INTERFACE I_Observable EXTENDS __SYSTEM.IQueryInterface

METHOD Attach : BOOL
VAR_INPUT
    ipObserver:         I_Observer;
END_VAR
END_METHOD

METHOD Detach : BOOL
VAR_INPUT
    ipObserver:         I_Observer;
END_VAR
END_METHOD

PROPERTY nObserverCount : UDINT
GET
END_GET
END_PROPERTY

METHOD Notify : I_Observable
VAR_INPUT
END_VAR
END_METHOD

METHOD NotifyLast : I_Observable
VAR_INPUT
END_VAR
END_METHOD

END_INTERFACE

(* stored: Version 1.1.0.1, ProductVersion 3.1.4024.12
   Itf I_Observable: Id {e9d5ee08-eb7e-494a-b197-8f922f772785}
   Method Attach: Id {30211a61-21d5-40ca-8122-c8c8f2acdb97}
   Method Detach: Id {ebccaf28-c550-4b56-881b-b9dc49898d61}
   Property nObserverCount: Id {07d52f56-10f6-4076-aab3-6b8ebc9310fa}
   Get Get: Id {3a19d823-a61c-41a4-83cb-832f68ece898}
   Method Notify: Id {dca0986e-fc2a-4198-a535-6eefd7c6a6f6}
   Method NotifyLast: Id {269f7bdd-fe70-43f6-bffb-4ca342e2c104} *)
